FUNCTION_BLOCK Clearing_State  IMPLEMENTS ITF_State
VAR_INPUT
END_VAR
VAR_OUTPUT
END_VAR
VAR
	pPML_Base : POINTER TO PML_Base;
	_stateMachine : IPmlStateMachine;
	bDone: BOOL;
END_VAR

{warning 'add method implementation '}
METHOD Cycle : BOOL
IF bDone THEN
	_stateMachine.SetStateComplete();
	pPML_Base^.SetState(pPML_Base^.stopped);
END_IF
END_METHOD

METHOD FB_init : BOOL
VAR_INPUT
	bInitRetains : BOOL; // if TRUE, the retain variables are initialized (warm start / cold start)
	bInCopyCode : BOOL;  // if TRUE, the instance afterwards gets moved into the copy code (online change)
	pPML_Base : POINTER TO PML_Base;
	statemachine : IPmlStateMachine;
END_VAR
_stateMachine := statemachine;
THIS^.pPML_Base := pPML_Base;
END_METHOD

END_FUNCTION_BLOCK

(* stored: Version 1.1.0.1, ProductVersion 3.1.4024.11
   POU Clearing_State: Id {c0e240cf-b21a-4849-856e-db4bf862a711}, SpecialFunc None
   Method Cycle: Id {3aaf4e1c-492f-4d94-91e7-90aee0cf7cf0}
   Method FB_init: Id {d64ba9be-88f5-479b-bc41-6f59705c9952} *)
